// Mitsubishi GX Works2 project: 타이머응용3   PLC: Q02/Q02H

PROGRAM MAIN
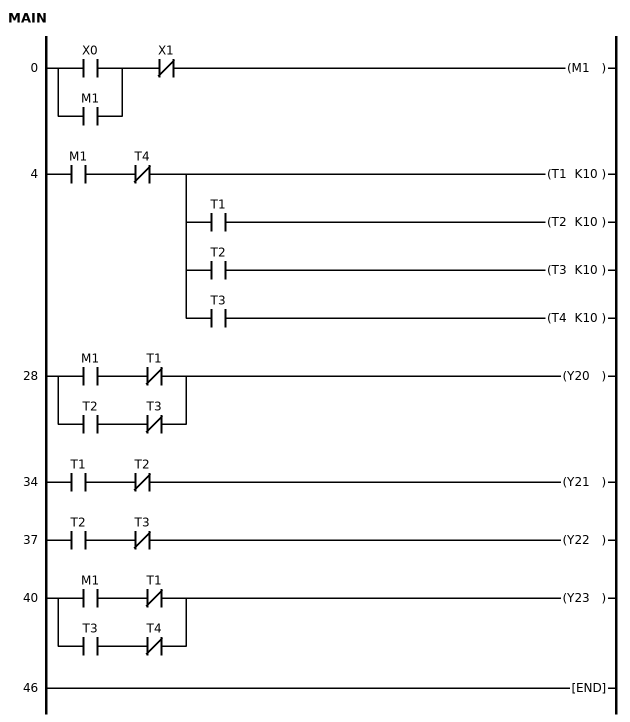
0     LD      X0
      OR      M1
      ANI     X1
      OUT     M1
4     LD      M1
      ANI     T4
      OUT     T1 K10
      MPS
      AND     T1
      OUT     T2 K10
      MRD
      AND     T2
      OUT     T3 K10
      MPP
      AND     T3
      OUT     T4 K10
28    LD      M1
      ANI     T1
      LD      T2
      ANI     T3
      ORB
      OUT     Y20
34    LD      T1
      ANI     T2
      OUT     Y21
37    LD      T2
      ANI     T3
      OUT     Y22
40    LD      M1
      ANI     T1
      LD      T3
      ANI     T4
      ORB
      OUT     Y23
46    END
END_PROGRAM
